// TIA Portal V18 export
// export: Created 2026-01-09T11:32:04.9535073Z, ExportSetting WithDefaults, DisplayName Totally Integrated Automation Portal, DisplayVersion V18 Update 5, DisplayName TIA Portal Openness, DisplayVersion V18 Update 5, DisplayName TIA Portal Teamcenter Gateway, DisplayVersion V18, DisplayName TIA Portal Version Control Interface, DisplayVersion V18, DisplayName SINAMICS Startdrive Advanced, DisplayVersion V18 SP2 Update 1, DisplayName SINAMICS Startdrive G110M, G120, G120C, G120D, G120P, G115D, DisplayVersion V18 SP2 Update 1, DisplayName SINAMICS Startdrive G130, G150, S120, S150, SINAMICS MV, S210, G220, S200, DisplayVersion V18 SP2 Update 1, DisplayName STEP 7 Professional, DisplayVersion V18 Update 5, DisplayName STEP 7 Safety, DisplayVersion V18, DisplayName WinCC Professional, DisplayVersion V18 Update 5
TagTable "Cylinder"
  CyVisual_Ctrl_End : Bool  (%DB[ST_CyDBNum].DBX134.3, CPU S71500-2PN_TP700, 1 s)
  CyVisual_Ctrl_Home : Bool  (%DB[ST_CyDBNum].DBX134.2, CPU S71500-2PN_TP700, 1 s)
  CyVisual_Ctrl_Next : Bool  (%DB[ST_CyDBNum].DBX134.1, CPU S71500-2PN_TP700, 1 s)
  CyVisual_Ctrl_Previous : Bool  (%DB[ST_CyDBNum].DBX134.0, CPU S71500-2PN_TP700, 1 s)
  CyVisual_Cy{4}_oHome(1) : Bool  (%DB[ST_CyDBNum].DBX32.3, CPU S71500-2PN_TP700, 1 s)
  CyVisual_CyPageNO : Int  (%DB[ST_CyDBNum].DBW128, CPU S71500-2PN_TP700, 1 s)
  CyVisual_CyTotalPageNO : Int  (%DB[ST_CyDBNum].DBW130, CPU S71500-2PN_TP700, 1 s)
  CyVisual_StructNum : Int  (%DB[ST_CyDBNum].DBW198, CPU S71500-2PN_TP700, 1 s)
  CyVisual_VisualAttribute{0} : Bool  (%DB[ST_CyDBNum].DBX196.0, CPU S71500-2PN_TP700, 1 s)
  CyVisual_VisualAttribute{1} : Bool  (%DB[ST_CyDBNum].DBX196.1, CPU S71500-2PN_TP700, 1 s)
  CyVisual_VisualAttribute{2} : Bool  (%DB[ST_CyDBNum].DBX196.2, CPU S71500-2PN_TP700, 1 s)
  CyVisual_VisualAttribute{3} : Bool  (%DB[ST_CyDBNum].DBX196.3, CPU S71500-2PN_TP700, 1 s)
  CyVisual_VisualAttribute{4} : Bool  (%DB[ST_CyDBNum].DBX196.4, CPU S71500-2PN_TP700, 1 s)
  ST_CyDBNum : Int  (1 s)
  STxxxCyHMIVisual_Cy{0}_GoHomeTime : Int  (%DB[ST_CyDBNum].DBW2, CPU S71500-2PN_TP700, 1 s)
  STxxxCyHMIVisual_Cy{0}_GoWorkTime : Int  (%DB[ST_CyDBNum].DBW4, CPU S71500-2PN_TP700, 1 s)
  STxxxCyHMIVisual_Cy{1}_GoHomeTime : Int  (%DB[ST_CyDBNum].DBW10, CPU S71500-2PN_TP700, 1 s)
  STxxxCyHMIVisual_Cy{1}_GoWorkTime : Int  (%DB[ST_CyDBNum].DBW12, CPU S71500-2PN_TP700, 1 s)
  STxxxCyHMIVisual_Cy{2}_GoHomeTime : Int  (%DB[ST_CyDBNum].DBW18, CPU S71500-2PN_TP700, 1 s)
  STxxxCyHMIVisual_Cy{2}_GoWorkTime : Int  (%DB[ST_CyDBNum].DBW20, CPU S71500-2PN_TP700, 1 s)
  STxxxCyHMIVisual_Cy{3}_GoHomeTime : Int  (%DB[ST_CyDBNum].DBW26, CPU S71500-2PN_TP700, 1 s)
  STxxxCyHMIVisual_Cy{3}_GoWorkTime : Int  (%DB[ST_CyDBNum].DBW28, CPU S71500-2PN_TP700, 1 s)
  STxxxCyHMIVisual_Cy{4}_GoHomeTime : Int  (%DB[ST_CyDBNum].DBW34, CPU S71500-2PN_TP700, 1 s)
  STxxxCyHMIVisual_Cy{4}_GoWorkTime : Int  (%DB[ST_CyDBNum].DBW36, CPU S71500-2PN_TP700, 1 s)
  CyVisual_Cy{1}_iWork : Bool  (%DB[ST_CyDBNum].DBX8.0, CPU S71500-2PN_TP700, 1 s)   // Cyl_02
  CyVisual_Cy{1}_iHome : Bool  (%DB[ST_CyDBNum].DBX8.1, CPU S71500-2PN_TP700, 1 s)   // Cyl_02
  CyVisual_Cy{4}_iHome : Bool  (%DB[ST_CyDBNum].DBX32.1, CPU S71500-2PN_TP700, 1 s)   // Cyl_05
  CyVisual_Cy{0}_oHomeInterlock : Bool  (%DB[ST_CyDBNum].DBX0.5, CPU S71500-2PN_TP700, 1 s)   // Cyl_01
  CyVisual_Cy{1}_oHomeInterlock : Bool  (%DB[ST_CyDBNum].DBX8.5, CPU S71500-2PN_TP700, 1 s)   // Cyl_02
  CyVisual_Cy{2}_ManualHome : Bool  (%DB[ST_CyDBNum].DBX22.1, CPU S71500-2PN_TP700, 1 s)   // Cyl_03
  CyVisual_Cy{3}_ManualWork : Bool  (%DB[ST_CyDBNum].DBX30.0, CPU S71500-2PN_TP700, 1 s)   // Cyl_04
  CyVisual_Cy{4}_oHome : Bool  (%DB[ST_CyDBNum].DBX32.3, CPU S71500-2PN_TP700, 1 s)   // Cyl_05
  CyVisual_Cy{2}_oHome : Bool  (%DB[ST_CyDBNum].DBX16.3, CPU S71500-2PN_TP700, 1 s)   // Cyl_03
  CyVisual_Cy{4}_oHomeInterlock : Bool  (%DB[ST_CyDBNum].DBX32.5, CPU S71500-2PN_TP700, 1 s)   // Cyl_05
  CyVisual_Cy{4}_owork : Bool  (%DB[ST_CyDBNum].DBX32.2, CPU S71500-2PN_TP700, 1 s)   // Cyl_05
  CyVisual_Cy{4}_iWork : Bool  (%DB[ST_CyDBNum].DBX32.0, CPU S71500-2PN_TP700, 1 s)   // Cyl_05
  CyVisual_Cy{0}_ManualWork : Bool  (%DB[ST_CyDBNum].DBX6.0, CPU S71500-2PN_TP700, 1 s)   // Cyl_01 DBX0.0
  CyVisual_Cy{3}_ManualHome : Bool  (%DB[ST_CyDBNum].DBX30.1, CPU S71500-2PN_TP700, 1 s)   // Cyl_04
  CyVisual_Cy{2}_oWorkInterlock : Bool  (%DB[ST_CyDBNum].DBX16.4, CPU S71500-2PN_TP700, 1 s)   // Cyl_03
  CyVisual_Cy{4}_CyNO : Byte  (%DB[ST_CyDBNum].DBB33, CPU S71500-2PN_TP700, 1 s)   // DBX400.0 for HMI
  CyVisual_Cy{0}_owork : Bool  (%DB[ST_CyDBNum].DBX0.2, CPU S71500-2PN_TP700, 1 s)   // Cyl_01
  CyVisual_Cy{4}_ManualWork : Bool  (%DB[ST_CyDBNum].DBX38.0, CPU S71500-2PN_TP700, 1 s)   // Cyl_05
  CyVisual_Cy{0}_CyNO : Byte  (%DB[ST_CyDBNum].DBB1, CPU S71500-2PN_TP700, 1 s)   // DBX400.0 for HMI
  CyVisual_Cy{3}_oHome : Bool  (%DB[ST_CyDBNum].DBX24.3, CPU S71500-2PN_TP700, 1 s)   // Cyl_04
  CyVisual_Cy{0}_oHome : Bool  (%DB[ST_CyDBNum].DBX0.3, CPU S71500-2PN_TP700, 1 s)   // Cyl_01
  CyVisual_Cy{2}_ManualWork : Bool  (%DB[ST_CyDBNum].DBX22.0, CPU S71500-2PN_TP700, 1 s)   // Cyl_03
  CyVisual_Cy{1}_ManualHome : Bool  (%DB[ST_CyDBNum].DBX14.1, CPU S71500-2PN_TP700, 1 s)   // Cyl_02
  CyVisual_Cy{1}_CyNO : Byte  (%DB[ST_CyDBNum].DBB9, CPU S71500-2PN_TP700, 1 s)   // DBX400.0 for HMI
  CyVisual_Cy{3}_oWorkInterlock : Bool  (%DB[ST_CyDBNum].DBX24.4, CPU S71500-2PN_TP700, 1 s)   // Cyl_04
  CyVisual_Cy{1}_ManualWork : Bool  (%DB[ST_CyDBNum].DBX14.0, CPU S71500-2PN_TP700, 1 s)   // Cyl_02
  CyVisual_Cy{2}_owork : Bool  (%DB[ST_CyDBNum].DBX16.2, CPU S71500-2PN_TP700, 1 s)   // Cyl_03
  CyVisual_Cy{2}_oHomeInterlock : Bool  (%DB[ST_CyDBNum].DBX16.5, CPU S71500-2PN_TP700, 1 s)   // Cyl_03
  CyVisual_Cy{3}_CyNO : Byte  (%DB[ST_CyDBNum].DBB25, CPU S71500-2PN_TP700, 1 s)   // DBX400.0 for HMI
  CyVisual_Cy{1}_oHome : Bool  (%DB[ST_CyDBNum].DBX8.3, CPU S71500-2PN_TP700, 1 s)   // Cyl_02
  CyVisual_Cy{3}_iHome : Bool  (%DB[ST_CyDBNum].DBX24.1, CPU S71500-2PN_TP700, 1 s)   // Cyl_04
  CyVisual_Cy{0}_iHome : Bool  (%DB[ST_CyDBNum].DBX0.1, CPU S71500-2PN_TP700, 1 s)   // Cyl_01
  CyVisual_Cy{4}_oWorkInterlock : Bool  (%DB[ST_CyDBNum].DBX32.4, CPU S71500-2PN_TP700, 1 s)   // Cyl_05
  CyVisual_Cy{4}_ManualHome : Bool  (%DB[ST_CyDBNum].DBX38.1, CPU S71500-2PN_TP700, 1 s)   // Cyl_05
  CyVisual_Cy{0}_ManualHome : Bool  (%DB[ST_CyDBNum].DBX6.1, CPU S71500-2PN_TP700, 1 s)   // Cyl_01
  CyVisual_Cy{3}_iWork : Bool  (%DB[ST_CyDBNum].DBX24.0, CPU S71500-2PN_TP700, 1 s)   // Cyl_04
  CyVisual_Cy{0}_oWorkInterlock : Bool  (%DB[ST_CyDBNum].DBX0.4, CPU S71500-2PN_TP700, 1 s)   // Cyl_01
  CyVisual_Cy{1}_owork : Bool  (%DB[ST_CyDBNum].DBX8.2, CPU S71500-2PN_TP700, 1 s)   // Cyl_02
  CyVisual_Cy{2}_iHome : Bool  (%DB[ST_CyDBNum].DBX16.1, CPU S71500-2PN_TP700, 1 s)   // Cyl_03
  CyVisual_Cy{0}_iWork : Bool  (%DB[ST_CyDBNum].DBX0.0, CPU S71500-2PN_TP700, 1 s)   // Cyl_01
  CyVisual_Cy{1}_oWorkInterlock : Bool  (%DB[ST_CyDBNum].DBX8.4, CPU S71500-2PN_TP700, 1 s)   // Cyl_02
  CyVisual_Cy{3}_oHomeInterlock : Bool  (%DB[ST_CyDBNum].DBX24.5, CPU S71500-2PN_TP700, 1 s)   // Cyl_04
  CyVisual_Cy{3}_owork : Bool  (%DB[ST_CyDBNum].DBX24.2, CPU S71500-2PN_TP700, 1 s)   // Cyl_04
  CyVisual_Cy{2}_iWork : Bool  (%DB[ST_CyDBNum].DBX16.0, CPU S71500-2PN_TP700, 1 s)   // Cyl_03
  CyVisual_Cy{2}_CyNO : Byte  (%DB[ST_CyDBNum].DBB17, CPU S71500-2PN_TP700, 1 s)   // DBX400.0 for HMI
